(****************************************************************************************)
(*							Beckhoff Automation Poland									*)
(*								L_TBGetBitOfByte v1.0									*)
(*									29.02.2007											*)
(*				This function returns the state of a single bit within a ”byte” value	*)
(*______________________________________________________________________________________*)
FUNCTION L_TBGetBitOfByte : BOOL
VAR_INPUT
	byInput: BYTE;
	byBitNr: BYTE;
END_VAR

CASE byBitNr OF
	0:
	L_TBGetBitOfByte := byInput.0;
	1:
	L_TBGetBitOfByte := byInput.1;
	2:
	L_TBGetBitOfByte := byInput.2;
	3:
	L_TBGetBitOfByte := byInput.3;
	4:
	L_TBGetBitOfByte := byInput.4;
	5:
	L_TBGetBitOfByte := byInput.5;
	6:
	L_TBGetBitOfByte := byInput.6;
	7:
	L_TBGetBitOfByte := byInput.7;
END_CASE

END_FUNCTION

(* stored: Version 1.1.0.1, ProductVersion 3.1.4026.13, FileIdentifier 74612ca53b6bd8829eaf43afe68696a5a25019e6, FileSignature 7768df1976c428c25b55223deacdc4f6652d482f32dbbc2ddca7c23b5453cb939694e225b7f1a44c1f96ff1f6f539f5d1b35ecf4e03fcdc7b917b24a60c7341ffcedd8607eaa497ceed6440ac7dac79653e0f49dd7ed593e0e4bed4a0da269263176d92ab1e9e4e4c58123e64186a933aa33da86f4bb86380d92cefe7dadd03d3cc1fb6c90d6d9640db88fda0f1eb079135ebaf64b18edf73d721a309574b34863607193718c2ebc561cbe11a323ab0110ccb1d20d9c366882faeca170f4311682741b0d808d01210542d2ffb303770f650ada643a927dfe10ce5fcf306c8acc7306a2cfd0052d7ab138b930b660f211eb8f368ff69cd50dc0ee6d215d1be156
   POU L_TBGetBitOfByte: Id {6d8a9ab6-e793-497e-b058-2dcbc09b33d7}, SpecialFunc None *)
